// Mitsubishi GX Works2 project: ZP_funtion_EX3   PLC: Q03UDV

PROGRAM MAIN
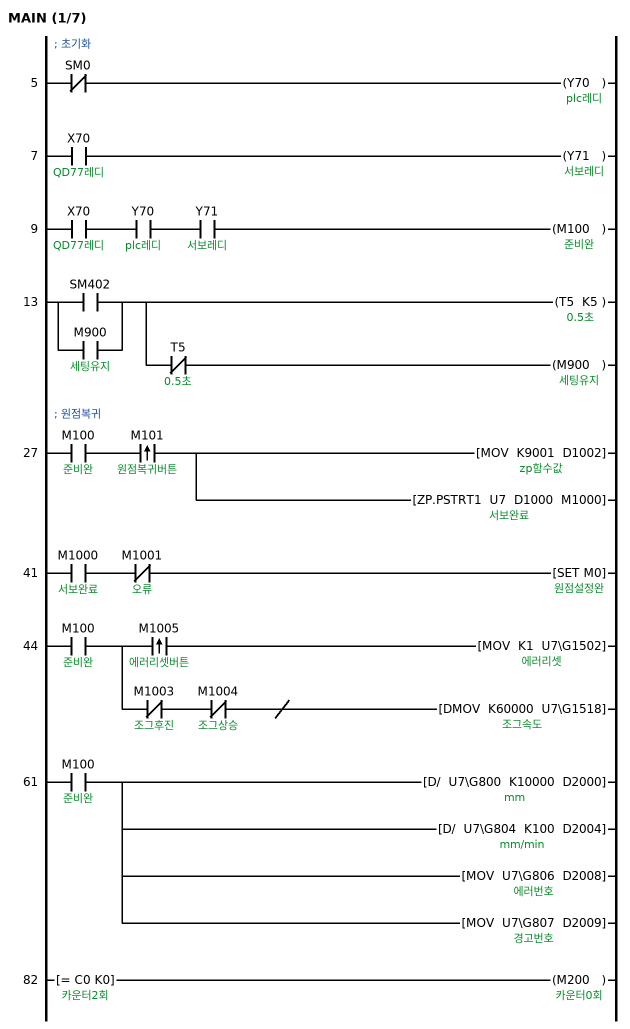
; 초기화
5     LDI     SM0
      OUT     Y70  ; plc레디
7     LD      X70  ; QD77레디
      OUT     Y71  ; 서보레디
9     LD      X70  ; QD77레디
      AND     Y70  ; plc레디
      AND     Y71  ; 서보레디
      OUT     M100  ; 준비완
13    LD      SM402
      OR      M900  ; 세팅유지
      OUT     T5 K5  ; 0.5초
      ANI     T5  ; 0.5초
      OUT     M900  ; 세팅유지
; 원점복귀
27    LD      M100  ; 준비완
      ANDP    M101  ; 원점복귀버튼
      MOV     K9001 D1002  ; zp함수값
      ZP.PSTRT1 U7 D1000 M1000  ; 서보완료
41    LD      M1000  ; 서보완료
      ANI     M1001  ; 오류
      SET     M0  ; 원점설정완
44    LD      M100  ; 준비완
      MPS
      ANDP    M1005  ; 에러리셋버튼
      MOV     K1 U7\G1502  ; 에러리셋
      MPP
      ANI     M1003  ; 조그후진
      ANI     M1004  ; 조그상승
      INV
      DMOV    K60000 U7\G1518  ; 조그속도
61    LD      M100  ; 준비완
      D/      U7\G800 K10000 D2000  ; mm
      D/      U7\G804 K100 D2004  ; mm/min
      MOV     U7\G806 D2008  ; 에러번호
      MOV     U7\G807 D2009  ; 경고번호
82    LD=     C0 K0  ; 카운터2회
      OUT     M200  ; 카운터0회
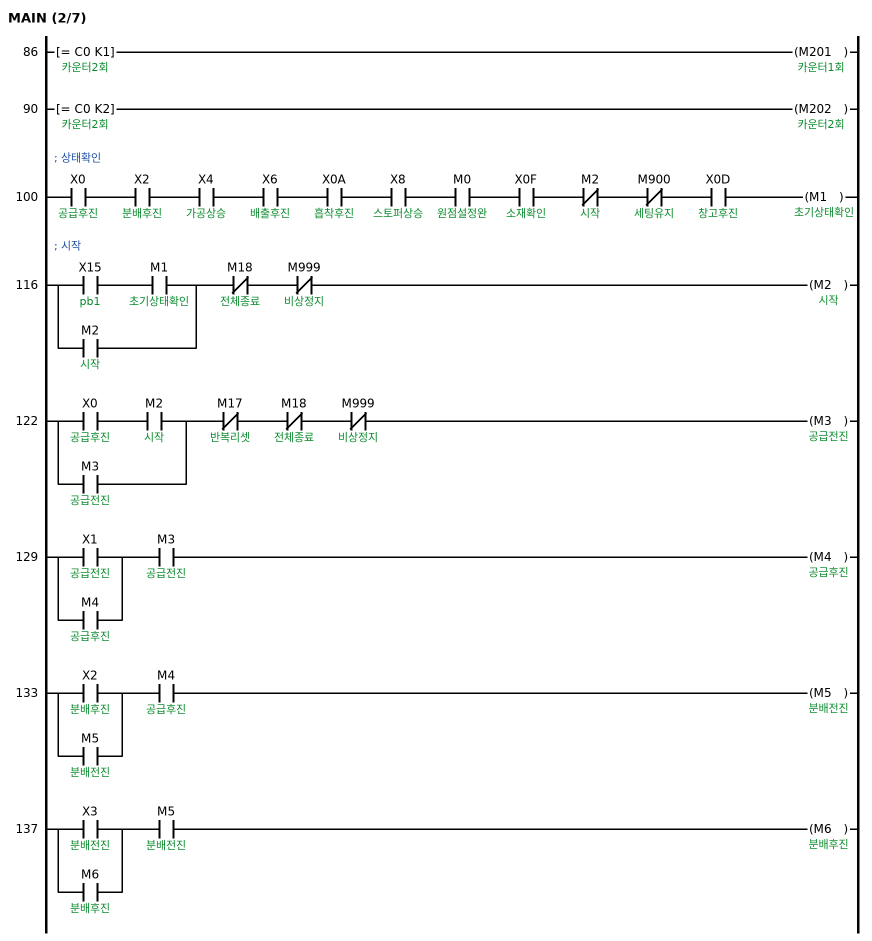
86    LD=     C0 K1  ; 카운터2회
      OUT     M201  ; 카운터1회
90    LD=     C0 K2  ; 카운터2회
      OUT     M202  ; 카운터2회
; 상태확인
100   LD      X0  ; 공급후진
      AND     X2  ; 분배후진
      AND     X4  ; 가공상승
      AND     X6  ; 배출후진
      AND     X0A  ; 흡착후진
      AND     X8  ; 스토퍼상승
      AND     M0  ; 원점설정완
      AND     X0F  ; 소재확인
      ANI     M2  ; 시작
      ANI     M900  ; 세팅유지
      AND     X0D  ; 창고후진
      OUT     M1  ; 초기상태확인
; 시작
116   LD      X15  ; pb1
      AND     M1  ; 초기상태확인
      OR      M2  ; 시작
      ANI     M18  ; 전체종료
      ANI     M999  ; 비상정지
      OUT     M2  ; 시작
122   LD      X0  ; 공급후진
      AND     M2  ; 시작
      OR      M3  ; 공급전진
      ANI     M17  ; 반복리셋
      ANI     M18  ; 전체종료
      ANI     M999  ; 비상정지
      OUT     M3  ; 공급전진
129   LD      X1  ; 공급전진
      OR      M4  ; 공급후진
      AND     M3  ; 공급전진
      OUT     M4  ; 공급후진
133   LD      X2  ; 분배후진
      OR      M5  ; 분배전진
      AND     M4  ; 공급후진
      OUT     M5  ; 분배전진
137   LD      X3  ; 분배전진
      OR      M6  ; 분배후진
      AND     M5  ; 분배전진
      OUT     M6  ; 분배후진
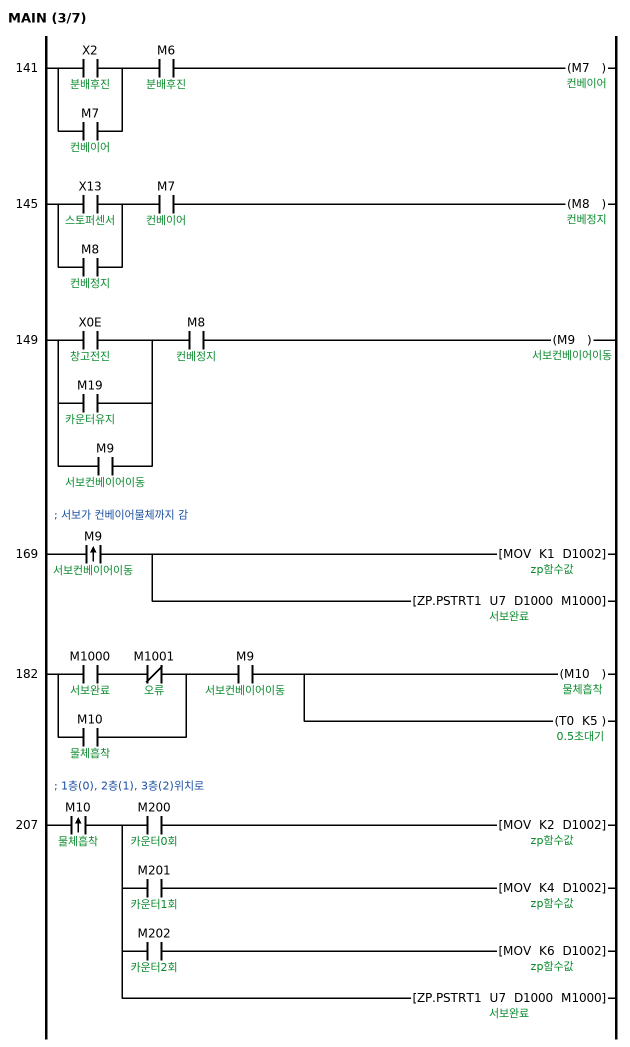
141   LD      X2  ; 분배후진
      OR      M7  ; 컨베이어
      AND     M6  ; 분배후진
      OUT     M7  ; 컨베이어
145   LD      X13  ; 스토퍼센서
      OR      M8  ; 컨베정지
      AND     M7  ; 컨베이어
      OUT     M8  ; 컨베정지
149   LD      X0E  ; 창고전진
      OR      M19  ; 카운터유지
      OR      M9  ; 서보컨베이어이동
      AND     M8  ; 컨베정지
      OUT     M9  ; 서보컨베이어이동
; 서보가 컨베이어물체까지 감
169   LDP     M9  ; 서보컨베이어이동
      MOV     K1 D1002
      ZP.PSTRT1 U7 D1000 M1000
182   LD      M1000  ; 서보완료
      ANI     M1001  ; 오류
      OR      M10  ; 물체흡착
      AND     M9  ; 서보컨베이어이동
      OUT     M10  ; 물체흡착
      OUT     T0 K5  ; 0.5초대기
; 1층(0), 2층(1), 3층(2)위치로
207   LDP     M10  ; 물체흡착
      MPS
      AND     M200  ; 카운터0회
      MOV     K2 D1002
      MRD
      AND     M201  ; 카운터1회
      MOV     K4 D1002
      MRD
      AND     M202  ; 카운터2회
      MOV     K6 D1002
      MPP
      ZP.PSTRT1 U7 D1000 M1000
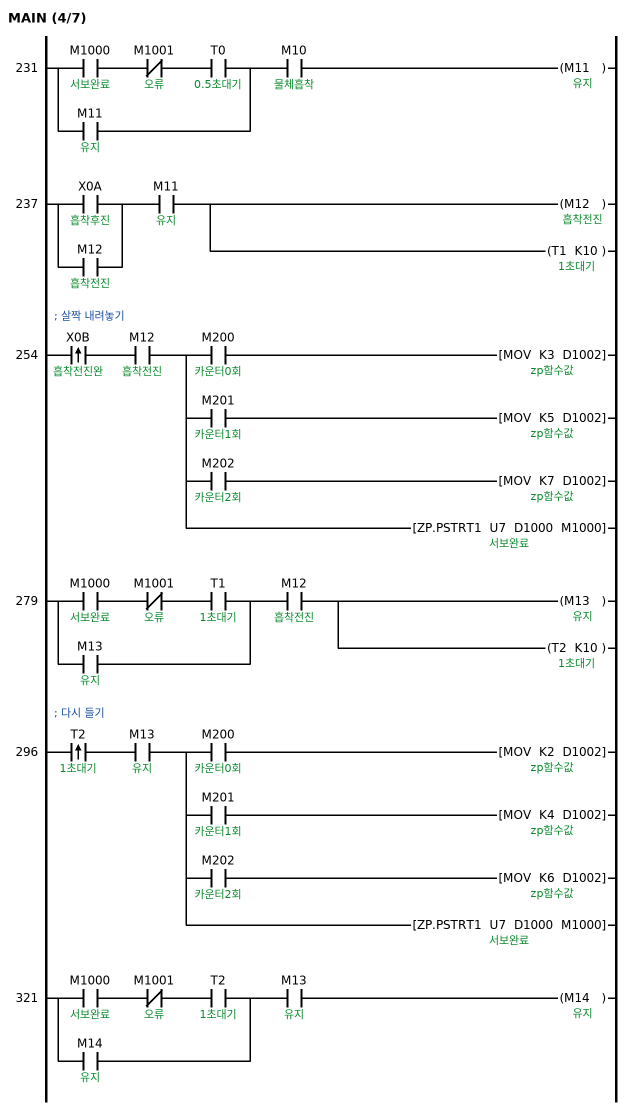
231   LD      M1000  ; 서보완료
      ANI     M1001  ; 오류
      AND     T0  ; 0.5초대기
      OR      M11  ; 유지
      AND     M10  ; 물체흡착
      OUT     M11  ; 유지
237   LD      X0A  ; 흡착후진
      OR      M12  ; 흡착전진
      AND     M11  ; 유지
      OUT     M12  ; 흡착전진
      OUT     T1 K10  ; 1초대기
; 살짝 내려놓기
254   LDP     X0B  ; 흡착전진완
      AND     M12  ; 흡착전진
      MPS
      AND     M200  ; 카운터0회
      MOV     K3 D1002
      MRD
      AND     M201  ; 카운터1회
      MOV     K5 D1002
      MRD
      AND     M202  ; 카운터2회
      MOV     K7 D1002
      MPP
      ZP.PSTRT1 U7 D1000 M1000
279   LD      M1000  ; 서보완료
      ANI     M1001  ; 오류
      AND     T1  ; 1초대기
      OR      M13  ; 유지
      AND     M12  ; 흡착전진
      OUT     M13  ; 유지
      OUT     T2 K10  ; 1초대기
; 다시 들기
296   LDP     T2  ; 1초대기
      AND     M13  ; 유지
      MPS
      AND     M200  ; 카운터0회
      MOV     K2 D1002
      MRD
      AND     M201  ; 카운터1회
      MOV     K4 D1002
      MRD
      AND     M202  ; 카운터2회
      MOV     K6 D1002
      MPP
      ZP.PSTRT1 U7 D1000 M1000
321   LD      M1000  ; 서보완료
      ANI     M1001  ; 오류
      AND     T2  ; 1초대기
      OR      M14  ; 유지
      AND     M13  ; 유지
      OUT     M14  ; 유지
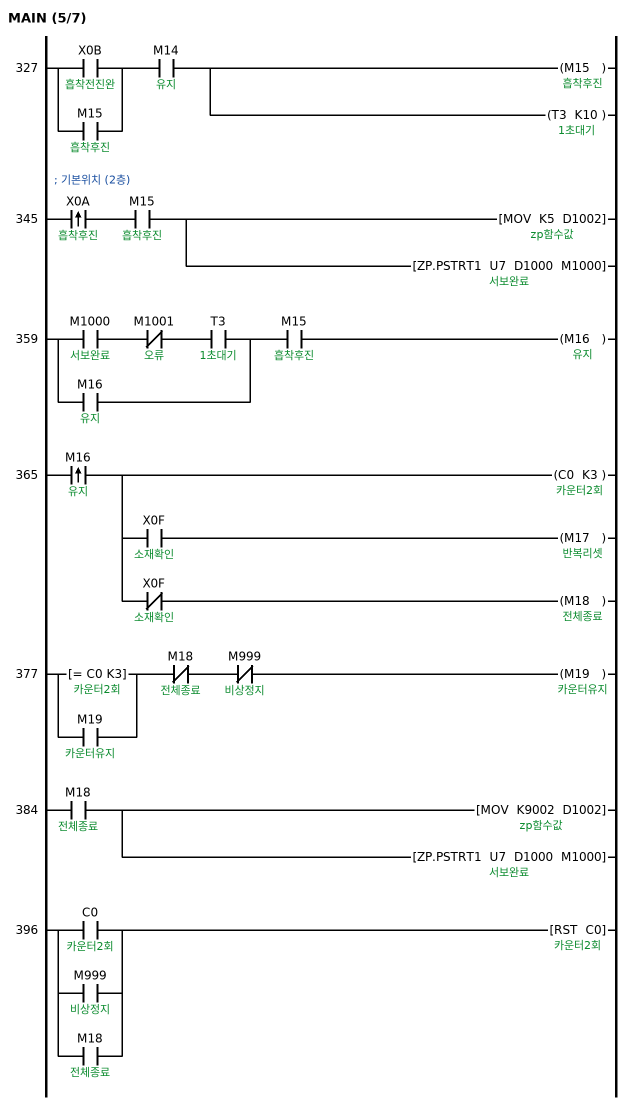
327   LD      X0B  ; 흡착전진완
      OR      M15  ; 흡착후진
      AND     M14  ; 유지
      OUT     M15  ; 흡착후진
      OUT     T3 K10  ; 1초대기
; 기본위치 (2층)
345   LDP     X0A  ; 흡착후진
      AND     M15  ; 흡착후진
      MOV     K5 D1002
      ZP.PSTRT1 U7 D1000 M1000
359   LD      M1000  ; 서보완료
      ANI     M1001  ; 오류
      AND     T3  ; 1초대기
      OR      M16  ; 유지
      AND     M15  ; 흡착후진
      OUT     M16  ; 유지
365   LDP     M16  ; 유지
      OUT     C0 K3  ; 카운터2회
      MPS
      AND     X0F  ; 소재확인
      OUT     M17  ; 반복리셋
      MPP
      ANI     X0F  ; 소재확인
      OUT     M18  ; 전체종료
377   LD=     C0 K3  ; 카운터2회
      OR      M19  ; 카운터유지
      ANI     M18  ; 전체종료
      ANI     M999  ; 비상정지
      OUT     M19  ; 카운터유지
384   LD      M18  ; 전체종료
      MOV     K9002 D1002
      ZP.PSTRT1 U7 D1000 M1000
396   LD      C0  ; 카운터2회
      OR      M999  ; 비상정지
      OR      M18  ; 전체종료
      RST     C0  ; 카운터2회
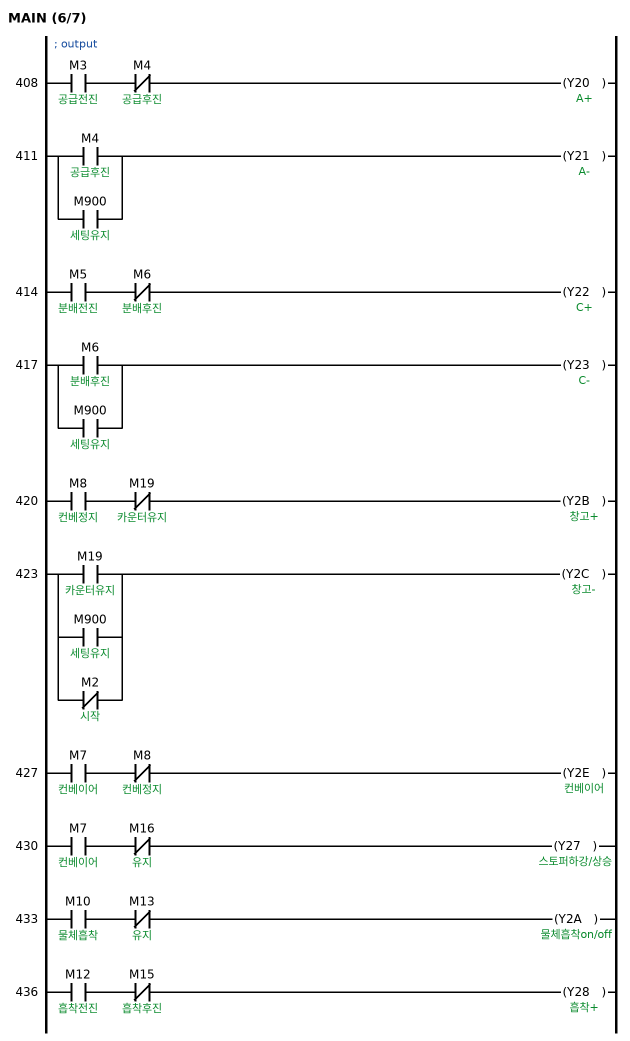
; output
408   LD      M3  ; 공급전진
      ANI     M4  ; 공급후진
      OUT     Y20  ; A+
411   LD      M4  ; 공급후진
      OR      M900  ; 세팅유지
      OUT     Y21  ; A-
414   LD      M5  ; 분배전진
      ANI     M6  ; 분배후진
      OUT     Y22  ; C+
417   LD      M6  ; 분배후진
      OR      M900  ; 세팅유지
      OUT     Y23  ; C-
420   LD      M8  ; 컨베정지
      ANI     M19  ; 카운터유지
      OUT     Y2B  ; 창고+
423   LD      M19  ; 카운터유지
      OR      M900  ; 세팅유지
      ORI     M2  ; 시작
      OUT     Y2C  ; 창고-
427   LD      M7  ; 컨베이어
      ANI     M8  ; 컨베정지
      OUT     Y2E  ; 컨베이어
430   LD      M7  ; 컨베이어
      ANI     M16  ; 유지
      OUT     Y27  ; 스토퍼하강/상승
433   LD      M10  ; 물체흡착
      ANI     M13  ; 유지
      OUT     Y2A  ; 물체흡착on/off
436   LD      M12  ; 흡착전진
      ANI     M15  ; 흡착후진
      OUT     Y28  ; 흡착+
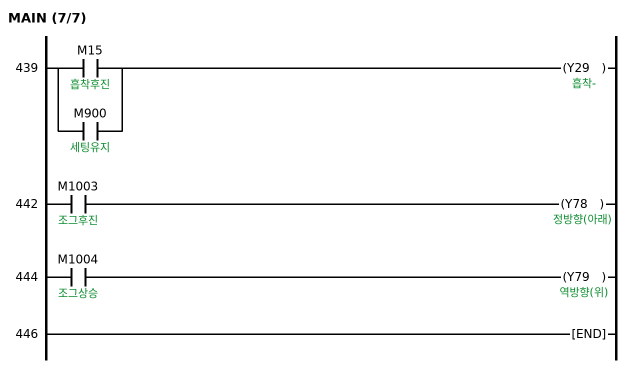
439   LD      M15  ; 흡착후진
      OR      M900  ; 세팅유지
      OUT     Y29  ; 흡착-
442   LD      M1003  ; 조그후진
      OUT     Y78  ; 정방향(아래)
444   LD      M1004  ; 조그상승
      OUT     Y79  ; 역방향(위)
446   END
END_PROGRAM

// device comments not shown above
M5000  ; 잠시막기
D2010  ; 경고번호
